INTERFACE PUBLIC I_MoveCommand EXTENDS AxisCommand

{attribute 'monitoring' := 'call'}
PROPERTY PUBLIC IsActive : BOOL
GET // PUBLIC
END_GET
END_PROPERTY

END_INTERFACE

(* stored: Version 1.1.0.1, ProductVersion 3.1.4026.13
   Itf I_MoveCommand: Id {b6727b9e-4791-0f05-1d47-70b23b903054}
   Property IsActive: Id {07dfa685-afcf-0682-382c-33a3c90ba725}
   Get Get: Id {d448bb17-d37c-025e-0194-0b48d05b973d} *)
